(* CoDeSys 2.3.9.41 project: 25_06_aspiNEW.pro *)
(* Libraries: STANDARD.LIB 4.10.05 11:14:46, IECSFC.LIB 13.4.06 15:51:28, ANALYZATION.LIB 5.10.99 09:05:06 *)

(* PLC configuration (modules and I/O channels)
xDI_Start_F1 AT %IX0.0 [BitInput] Discrete input 1 {ChannellName = Enter name}
xDI_Stop_F1 AT %IX0.1 [BitInput] Discrete input 2 {ChannellName = Enter name}
xDI_Start_F2 AT %IX0.2 [BitInput] Discrete input 3 {ChannellName = Enter name}
xDI_Stop_F2 AT %IX0.3 [BitInput] Discrete input 4 {ChannellName = Enter name}
AT %IB1.0 [ByteInput] 8 discrete inputs {ChannellName = Enter name}
AT %IB1.1 [ByteInput] 8 discrete inputs {ChannellName = Enter name}
AT %IB1.2 [ByteInput] 8 discrete inputs {ChannellName = Enter name}
AT %IB1.3 [ByteInput] 8 discrete inputs {ChannellName = Enter name}
AT %QX2.0 [BitOutput] Fast discrete output 1 {ChannellName = Enter name}
AT %QX2.1 [BitOutput] Fast discrete output 2 {ChannellName = Enter name}
AT %QX2.2 [BitOutput] Fast discrete output 3 {ChannellName = Enter name}
xDO_Lamp_F1 AT %QX2.3 [BitOutput] Fast discrete output 4 {ChannellName = Enter name}
AT %QB3.0 [ByteOutput] 8 discrete outputs {ChannellName = Enter name}
AT %QB3.1 [ByteOutput] 8 discrete outputs {ChannellName = Enter name}
AT %QB3.2 [ByteOutput] 4 discrete outputs {ChannellName = Enter name}
Special input [ID103] node 4, in %IB4 out %QB4 {ChannellName = Special input}
  AT %IX4.0 [BitInput] Special input {ChannellName = Enter name}
Special output [ID104] node 5, in %IB5 out %QB5 {ChannellName = Special output}
  AT %QX5.0 [BitOutput] Special output {ChannellName = Enter name}
TCP [TCP_ID221] node 0, in %IB6.0.0 out %QB6.0.0 {ChannellName = TCP; RemotePort = 502; Visibility = No}
AT %QB6.1.0 [ByteOutput] {ChannellName = Enter name}
AT %QB6.2.0 [ByteOutput] {ChannellName = Enter name}
AT %QB6.3.0 [ByteOutput] {ChannellName = Enter name}
AT %QB6.4.0 [ByteOutput] {ChannellName = Enter name}
AT %QB6.5.0 [ByteOutput] {ChannellName = Enter name}
AT %QB6.6.0 [ByteOutput] {ChannellName = Enter name}
AT %QB6.7.0 [ByteOutput] {ChannellName = Enter name}
uiDelay_SCR_s AT %QW6.8.0 [WordOutput] {ChannellName = Enter name}
uiDelay_FAN_s AT %QW6.9.0 [WordOutput] {ChannellName = Enter name}
uiVib_Work_s AT %QW6.10.0 [WordOutput] {ChannellName = Enter name}
uiVib_Pause_min AT %QW6.11.0 [WordOutput] {ChannellName = Enter name}
uiHatch_Max_s AT %QW6.12.0 [WordOutput] {ChannellName = Enter name}
uiDrive_SpeedTimeout_s AT %QW6.13.0 [WordOutput] {ChannellName = Enter name}
uiFansRunning AT %QW6.14.0 [WordOutput] {ChannellName = Enter name}
uiModeDisplay AT %QW6.15.0 [WordOutput] {ChannellName = Enter name}
*)

(* Global variable list: GVL_AlarmIdx *)
VAR_GLOBAL CONSTANT
	ALM_EMERGENCY       : INT := 1;
	ALM_PRESSURE        : INT := 2;
	ALM_TF_DRIVE        : INT := 3;
	ALM_EXHAUST_DRIVE   : INT := 4;
	ALM_SCR_DRIVE       : INT := 5;
	ALM_SCR_IMPOSSIBLE  : INT := 7;
	ALM_F1_DRIVE        : INT := 10;
	ALM_F2_DRIVE        : INT := 11;
	ALM_F3_DRIVE        : INT := 12;
	ALM_F4_DRIVE        : INT := 13;
	ALM_F5_DRIVE        : INT := 14;
	ALM_VIB1            : INT := 20;
	ALM_VIB2            : INT := 21;
	ALM_HATCH 		: INT := 22;
	ALM_HATCH_TIMEOUT   : INT := 23;
END_VAR

(* Global variable list: GVL_App *)
VAR_GLOBAL
	(* === Исполнительные механизмы === *)
	TF		: ST_Motor;					(* Транспортный вентилятор *)
	Exhaust : ST_Motor;					(*Вытяжка*)
	SCR		: ST_Motor;					(* Шнек *)
	Fans	: ARRAY[1..5] OF ST_Fan;	(* Вентиляторы станков 1..5 *)
	Vib		: ST_Vibrator;				(* Пара вибраторов *)
	Hatch	: ST_Hatch;					(* Люк *)
	
	(* === Состояние системы === *)
	Alarms		: ST_Alarms;
	xModeManual	: BOOL;		(* Режим: FALSE = автомат, TRUE = ручной *)
	xAckAlarm	: BOOL;		(* Квитирование аварии (с панели) *)
	xMasterOK	: BOOL;		(* Магистраль готова (ТВ + шнек работают штатно) *)
END_VAR

(* Global variable list: GVL_HMI *)
VAR_GLOBAL RETAIN
	Settings : ST_Settings := (
		uiDelay_SCR_s          := 5,
		uiDelay_FAN_s          := 3,
		uiVib_Work_s           := 10,
		uiVib_Pause_min        := 30,
		uiHatch_Max_s          := 30,
		uiDrive_SpeedTimeout_s := 15	(* НОВОЕ *)
	);
END_VAR

(* Global variable list: GVL_Test *)
VAR_GLOBAL
	(* === Аварии === *)
	mb_Emergency      : BOOL;
	mb_Pressure       : BOOL;
	mb_TF_Alarm       : BOOL;
	mb_Exhaust_Alarm  : BOOL;
	mb_SCR_Alarm      : BOOL;
	mb_SCR_Impossible : BOOL;
	mb_Fan1_Alarm  : BOOL;
	mb_Fan2_Alarm  : BOOL;
	mb_Fan3_Alarm  : BOOL;
	mb_Fan4_Alarm  : BOOL;
	mb_Fan5_Alarm  : BOOL;
	mb_Vib1_Alarm  : BOOL;
	mb_Vib2_Alarm  : BOOL;
	mb_Hatch_Alarm   : BOOL;
	mb_Hatch_Timeout : BOOL;
END_VAR

(* Data type *)
TYPE E_DriveState :
(
	DRIVE_STOPPED  := 0,
	DRIVE_STARTING := 1,
	DRIVE_RUNNING  := 2,
	DRIVE_STOPPING := 3,
	DRIVE_FAULT    := 10
);
END_TYPE

(* Data type *)
TYPE E_HatchState :
(
	HATCH_UNKNOWN := 0,
	HATCH_CLOSED  := 1,
	HATCH_OPENING := 2,
	HATCH_OPEN    := 3,
	HATCH_CLOSING := 4,
	HATCH_FAULT   := 10
);
END_TYPE

(* Data type *)
TYPE E_VibState :
(
	VIB_IDLE	:= 0,	(* Выключено (xEnable=FALSE) *)
	VIB_PAUSE	:= 1,	(* Пауза между циклами *)
	VIB_WORK	:= 2	(* Фаза работы *)
);
END_TYPE

(* Data type *)
TYPE ST_Alarms :
STRUCT
	(* Критические *)
	xEmergencyStop  : BOOL;
	xPressure       : BOOL;
	xTF_Alarm       : BOOL;
	xExhaust_Alarm  : BOOL;
	xSCR_Alarm      : BOOL;
	xSCR_Impossible : BOOL;
	(* Предупреждения *)
	axFan_Alarm     : ARRAY[1..5] OF BOOL;
	xVib1_Alarm     : BOOL;
	xVib2_Alarm     : BOOL;
	xHatch_Alarm : BOOL;
	xHatch_Timeout  : BOOL;
	(* Обобщённые *)
	xAny      : BOOL;
	xCritical : BOOL;
	xWarning  : BOOL;
END_STRUCT
END_TYPE

(* Data type *)
TYPE ST_Fan :
STRUCT
    (* === Команды (вход в FB) === *)
 	xCmdStart    : BOOL;    (* Команда пуска (с кнопки или с панели) *)
	xCmdStop     : BOOL;    (* Команда стопа *)

	(* === Сигналы с поля (вход в FB) === *)
	xReady       : BOOL;    (* "Готов" от частотника (DI_readyF1) *)
	xAtSpeed  : BOOL;    (* "Авария" от частотника (DI_alarmF1) *)

	(* === Выход на ИМ === *)
	xRun         : BOOL;    (* Команда на пуск частотника (DO_F1) *)

	(* === Состояние (выход FB) === *)
	xEnabled     : BOOL;    (* Зафиксирован запрос на работу (был xFlag1) *)
	xFault       : BOOL;    (* Обобщённая неисправность (заменяет F1_OFF) *)
	eState       : E_DriveState;  (* Состояние машины: Stopped/Starting/Running/Fault *)

	(* === Статистика === *)
	udiStarts    : UDINT;   (* Счётчик пусков *)
	rHours       : REAL;    (* Моточасы *)
END_STRUCT
END_TYPE

(* Data type *)
TYPE ST_Hatch :
STRUCT
	(* === Команды === *)
	xCmdOpen      : BOOL;	(* Команда "Открыть" (удержание) *)
	xCmdClose     : BOOL;	(* Команда "Закрыть" (удержание) *)

	(* === Сигналы с поля === *)
	xLS_Open      : BOOL;	(* Концевик "Открыт" (DI33) *)
	xLS_Closed    : BOOL;	(* Концевик "Закрыт" (DI34) *)
	xAlarmHM      : BOOL;	(* Авария двигателя шибера (DI31) *)

	(* === Выходы на ИМ === *)
	xOpen         : BOOL;	(* DO "Открыть" (DO18) *)
	xClose        : BOOL;	(* DO "Закрыть" (DO19) *)

	(* === Состояние === *)
	eState        : E_HatchState;
	xFaultTimeout : BOOL;	(* Заклинило — таймаут *)
	xFault        : BOOL;	(* Обобщённая *)
END_STRUCT
END_TYPE

(* Data type *)
TYPE ST_Motor :
STRUCT
	(* === Команды (вход в FB) === *)
	xCmdRun		: BOOL;		(* Запрос на работу от секвенсора *)
	
	(* === Сигналы с поля === *)
	xReady		: BOOL;		(* "Готов" от частотника *)
	xAtSpeed	: BOOL;		(* "Авария" от частотника *)
	xRotation	: BOOL;		(* Импульсы датчика вращения (только для шнека) *)
	
	(* === Выход на ИМ === *)
	xRun		: BOOL;		(* Команда на пуск частотника *)
	
	(* === Состояние === *)
	xFault		: BOOL;		(* Обобщённая неисправность *)
	xNoRotation	: BOOL;		(* Авария "Не вращается" (только для шнека) *)
	eState		: E_DriveState;
END_STRUCT
END_TYPE

(* Data type *)
TYPE ST_Settings :
STRUCT
	(* === Тайминги секвенсора, секунды === *)
	uiDelay_SCR_s		: UINT;		(* Задержка пуска шнека после ТВ *)
	uiDelay_FAN_s		: UINT;		(* Задержка пуска вентилятора после шнека *)
	
	(* === Тайминги вибраторов === *)
	uiVib_Work_s		: UINT;		(* Длительность работы, секунды *)
	uiVib_Pause_min		: UINT;		(* Пауза между циклами, минуты *)
	
	(* === Тайминги люка === *)
	uiHatch_Max_s		: UINT;		(* Макс. время хода до концевика, секунды *)
	
	(* === Контроль шнека === *)
	uiScr_Window_s		: UINT;		(* Окно контроля вращения, секунды *)
	uiScr_PulseMin		: UINT;		(* Мин. импульсов за окно *)

	uiDrive_SpeedTimeout_s : UINT;
END_STRUCT
END_TYPE

(* Data type *)
TYPE ST_Vibrator :
STRUCT
	(* === Команды === *)
	xEnable		: BOOL;		(* Разрешение работы (от секвенсора: шнек работает) *)
	
	(* === Сигналы с поля === *)
	xAlarmV1	: BOOL;		(* Авария вибратора 1 *)
	xAlarmV2	: BOOL;		(* Авария вибратора 2 *)
	
	(* === Выходы на ИМ === *)
	xRunV1		: BOOL;
	xRunV2		: BOOL;
	
	(* === Состояние === *)
	xFault		: BOOL;
	xActive		: BOOL;		(* Сейчас идёт фаза работы (не паузы) *)
END_STRUCT
END_TYPE

(* POU PLC_PRG, ST *)
PROGRAM PLC_PRG
VAR
	(* === FB основных механизмов === *)
	FB_TF       : FB_Motor;
	FB_Exhaust  : FB_Motor;
	FB_SCR      : FB_Motor;
	FB_Fans     : ARRAY[1..5] OF FB_Fan;
	FB_Hatch    : FB_Hatch;
	FB_Vibrator : FB_Vibrator;
	FB_Alarms   : ARRAY[1..30] OF FB_Alarm;

	(* === Таймеры === *)
	TON_SCR_Delay : TON;
	TON_SCR_OffDelay : TON;	(* задержка выключения шнека *)
	TON_TF_OffDelay  : TON;	(* задержка выключения ТВ *)
	xAnyFanEnabled   : BOOL;	(* есть хоть один запрошенный вентилятор *)

	(* === Локальные массивы-агрегаторы команд === *)
	axCmdStart   : ARRAY[1..5] OF BOOL;
	axCmdStop    : ARRAY[1..5] OF BOOL;
	(*axAlarmDrive : ARRAY[1..5] OF BOOL;*)
	axAtSpeed :ARRAY[1..5] OF BOOL;
	axHMI_Man_Fan : ARRAY[1..5] OF BOOL;

	(* === Индекс цикла === *)
	i : INT;

	(* === Локальные копии TIME-настроек === *)
	tFanDelay  : TIME;
	tScrDelay  : TIME;
	tHatchMax  : TIME;
	tVibWork   : TIME;
	tVibPause  : TIME;
	tSpeedTimeout : TIME;

	(* === Флаги взаимной блокировки шибер <-> ИМ === *)
	xHatchClosed : BOOL;
	xAllStopped  : BOOL;

	xSettingsInit : BOOL;

	TON_Blink1 : TON;
	TON_Blink2 : TON;
	xBlink     : BOOL;
END_VAR
Inputs();
Diagnostics();
Sequence();
Outputs();
HMI();
ModbusMap();
END_PROGRAM
ACTION Diagnostics:
(* === КРИТИЧЕСКИЕ === *)
FB_Alarms[ALM_EMERGENCY](xCause := xDI_AlarmRelay, xAck := xAckAlarm);
Alarms.xEmergencyStop := FB_Alarms[ALM_EMERGENCY].xActive;

(* НЗ-контакт: норма = 24В (TRUE), авария/обрыв = нет 24В (FALSE) *)
FB_Alarms[ALM_PRESSURE](xCause := NOT xDI_Pressure, xAck := xAckAlarm);
Alarms.xPressure := FB_Alarms[ALM_PRESSURE].xActive;

(*FB_Alarms[ALM_TF_DRIVE](xCause := xDI_Alarm_TF, xAck := xAckAlarm);*)
FB_Alarms[ALM_TF_DRIVE](xCause := TF.xFault, xAck := xAckAlarm);
Alarms.xTF_Alarm := FB_Alarms[ALM_TF_DRIVE].xActive;

FB_Alarms[ALM_EXHAUST_DRIVE](xCause := xDI_Alarm_Exhaust, xAck := xAckAlarm);
Alarms.xExhaust_Alarm := FB_Alarms[ALM_EXHAUST_DRIVE].xActive;

(*FB_Alarms[ALM_SCR_DRIVE](xCause := xDI_Alarm_SCR, xAck := xAckAlarm);*)
FB_Alarms[ALM_SCR_DRIVE](xCause := SCR.xFault, xAck := xAckAlarm);
Alarms.xSCR_Alarm := FB_Alarms[ALM_SCR_DRIVE].xActive;

FB_Alarms[ALM_SCR_IMPOSSIBLE](xCause := NOT xDI_SCR_Impossible, xAck := xAckAlarm);
Alarms.xSCR_Impossible := FB_Alarms[ALM_SCR_IMPOSSIBLE].xActive;

(* === ВЕНТИЛЯТОРЫ 1..5 === *)
FB_Alarms[ALM_F1_DRIVE](xCause := Fans[1].xFault, xAck := xAckAlarm);
FB_Alarms[ALM_F2_DRIVE](xCause := Fans[2].xFault, xAck := xAckAlarm);
FB_Alarms[ALM_F3_DRIVE](xCause := Fans[3].xFault, xAck := xAckAlarm);
FB_Alarms[ALM_F4_DRIVE](xCause := Fans[4].xFault, xAck := xAckAlarm);
FB_Alarms[ALM_F5_DRIVE](xCause := Fans[5].xFault, xAck := xAckAlarm);

Alarms.axFan_Alarm[1] := FB_Alarms[ALM_F1_DRIVE].xActive;
Alarms.axFan_Alarm[2] := FB_Alarms[ALM_F2_DRIVE].xActive;
Alarms.axFan_Alarm[3] := FB_Alarms[ALM_F3_DRIVE].xActive;
Alarms.axFan_Alarm[4] := FB_Alarms[ALM_F4_DRIVE].xActive;
Alarms.axFan_Alarm[5] := FB_Alarms[ALM_F5_DRIVE].xActive;

(* === ВИБРАТОРЫ === *)
FB_Alarms[ALM_VIB1](xCause := xDI_Alarm_V1, xAck := xAckAlarm);
Alarms.xVib1_Alarm := FB_Alarms[ALM_VIB1].xActive;

FB_Alarms[ALM_VIB2](xCause := xDI_Alarm_V2, xAck := xAckAlarm);
Alarms.xVib2_Alarm := FB_Alarms[ALM_VIB2].xActive;

(* === ШИБЕР === *)
FB_Alarms[ALM_HATCH](xCause := xDI_Alarm_Hatch, xAck := xAckAlarm);
Alarms.xHatch_Alarm := FB_Alarms[ALM_HATCH].xActive;

FB_Alarms[ALM_HATCH_TIMEOUT](xCause := Hatch.xFaultTimeout, xAck := xAckAlarm);
Alarms.xHatch_Timeout := FB_Alarms[ALM_HATCH_TIMEOUT].xActive;

(* === КРИТИЧНЫЕ аварии: запрещают пуск всего, красный + зуммер === *)
Alarms.xCritical :=
	Alarms.xEmergencyStop                  (* аварийный стоп *)
	OR Alarms.xPressure                    (* нет разрежения *)
	OR Alarms.xSCR_Impossible              (* переполнение шнека *)
	OR FB_Alarms[ALM_TF_DRIVE].xActive     (* ТВ не набрал обороты — критично *)
	OR FB_Alarms[ALM_SCR_DRIVE].xActive;   (* шнек не набрал обороты — критично *)

(* === ПРЕДУПРЕЖДЕНИЯ: некритичные, жёлтый, система работает === *)
Alarms.xWarning :=
	FB_Alarms[ALM_F1_DRIVE].xActive
	OR FB_Alarms[ALM_F2_DRIVE].xActive
	OR FB_Alarms[ALM_F3_DRIVE].xActive
	OR FB_Alarms[ALM_F4_DRIVE].xActive
	OR FB_Alarms[ALM_F5_DRIVE].xActive
	OR FB_Alarms[ALM_VIB1].xActive
	OR FB_Alarms[ALM_VIB2].xActive
	OR FB_Alarms[ALM_HATCH].xActive;

Alarms.xAny := Alarms.xCritical OR Alarms.xWarning;

(* === СВЕТОФОР И ЗУММЕР === *)
IF Alarms.xCritical THEN
	xDO_Green  := FALSE;
	xDO_Yellow := FALSE;
	xDO_Red    := TRUE;
	xDO_Buzzer := TRUE;
ELSIF Alarms.xWarning OR NOT xDI_LS_Closed THEN
	xDO_Green  := FALSE;
	xDO_Yellow := TRUE;
	xDO_Red    := FALSE;
	xDO_Buzzer := FALSE;
ELSE
	xDO_Green  := TRUE;
	xDO_Yellow := FALSE;
	xDO_Red    := FALSE;
	xDO_Buzzer := FALSE;
END_IF
END_ACTION
ACTION HMI:
(* Сброс импульсных команд (кнопки вентиляторов) *)
xHMI_Start_F1 := FALSE;
xHMI_Start_F2 := FALSE;
xHMI_Start_F3 := FALSE;
xHMI_Start_F4 := FALSE;
xHMI_Start_F5 := FALSE;

xHMI_Stop_F1 := FALSE;
xHMI_Stop_F2 := FALSE;
xHMI_Stop_F3 := FALSE;
xHMI_Stop_F4 := FALSE;
xHMI_Stop_F5 := FALSE;

xHMI_AckAlarm := FALSE;
END_ACTION
ACTION Inputs:
(* Управление вентиляторами *)
axCmdStart[1] := xDI_Start_F1 OR xHMI_Start_F1;
axCmdStart[2] := xDI_Start_F2 OR xHMI_Start_F2;
axCmdStart[3] := xDI_Start_F3 OR xHMI_Start_F3;
axCmdStart[4] := xDI_Start_F4 OR xHMI_Start_F4;
axCmdStart[5] := xDI_Start_F5 OR xHMI_Start_F5;

axCmdStop[1] := xDI_Stop_F1 OR xHMI_Stop_F1;
axCmdStop[2] := xDI_Stop_F2 OR xHMI_Stop_F2;
axCmdStop[3] := xDI_Stop_F3 OR xHMI_Stop_F3;
axCmdStop[4] := xDI_Stop_F4 OR xHMI_Stop_F4;
axCmdStop[5] := xDI_Stop_F5 OR xHMI_Stop_F5;

(* Аварии частотников вентиляторов *)
(*
axAlarmDrive[1] := xDI_Alarm_F1;
axAlarmDrive[2] := xDI_Alarm_F2;
axAlarmDrive[3] := xDI_Alarm_F3;
axAlarmDrive[4] := xDI_Alarm_F4;
axAlarmDrive[5] := xDI_Alarm_F5;
*)

axAtSpeed[1] := xDI_AtSpeed_F1;
axAtSpeed[2] := xDI_AtSpeed_F2;
axAtSpeed[3] := xDI_AtSpeed_F3;
axAtSpeed[4] := xDI_AtSpeed_F4;
axAtSpeed[5] := xDI_AtSpeed_F5;

(* Команды на шибер *)
IF xModeManual THEN
	Hatch.xCmdOpen  := xHMI_Man_Open;
	Hatch.xCmdClose := xHMI_Man_Close;
ELSE
	Hatch.xCmdOpen  := xDI_Open  OR xHMI_Open;
	Hatch.xCmdClose := xDI_Close OR xHMI_Close;
END_IF

(* Сервисные сигналы *)
xAckAlarm   := xHMI_AckAlarm;
xModeManual := xHMI_ModeManual;

(* Ручные toggle вентиляторов -> в массив для цикла *)
axHMI_Man_Fan[1] := xHMI_Man_F1;
axHMI_Man_Fan[2] := xHMI_Man_F2;
axHMI_Man_Fan[3] := xHMI_Man_F3;
axHMI_Man_Fan[4] := xHMI_Man_F4;
axHMI_Man_Fan[5] := xHMI_Man_F5;
END_ACTION
ACTION ModbusMap:
(* ============================================================
   Action: ModbusMap — "промежуточные реле" для Modbus
   Копирование значений из структур в плоские переменные,
   т.к. конфигуратор ПЛК 2.3 не привязывает поля структур.
   Только ЧТЕНИЕ структур -> запись в mb_* (состояния на панель).
   ============================================================ *)

(* В начало ModbusMap *)
IF NOT xSettingsInit THEN
	IF uiDelay_SCR_s = 0 AND uiDelay_FAN_s = 0 THEN
		uiDelay_SCR_s   := 5;
		uiDelay_FAN_s   := 3;
		uiVib_Work_s    := 10;
		uiVib_Pause_min := 30;
		uiHatch_Max_s   := 30;
	END_IF
	xSettingsInit := TRUE;
END_IF

(* Работа механизмов *)
mb_Fan1_Run    := Fans[1].xRun;
mb_Fan2_Run    := Fans[2].xRun;
mb_Fan3_Run    := Fans[3].xRun;
mb_Fan4_Run    := Fans[4].xRun;
mb_Fan5_Run    := Fans[5].xRun;
mb_TF_Run      := TF.xRun;
mb_SCR_Run     := SCR.xRun;
mb_Exhaust_Run := Exhaust.xRun;

(* Вибраторы, магистраль, концевики *)
mb_Vib1_Run    := Vib.xRunV1;
mb_Vib2_Run    := Vib.xRunV2;
mb_Vib_Active  := Vib.xActive;
mb_MasterOK    := xMasterOK;
mb_LS_Open     := xDI_LS_Open;
mb_LS_Closed   := xDI_LS_Closed;
mb_Hatch_Open  := Hatch.xOpen;
mb_Hatch_Close := Hatch.xClose;

(* Аварии *)
mb_Emergency      := Alarms.xEmergencyStop;
mb_Pressure       := Alarms.xPressure;
mb_TF_Alarm       := Alarms.xTF_Alarm;
mb_Exhaust_Alarm  := Alarms.xExhaust_Alarm;
mb_SCR_Alarm      := Alarms.xSCR_Alarm;
mb_SCR_Impossible := Alarms.xSCR_Impossible;
mb_Fan1_Alarm  := Alarms.axFan_Alarm[1];
mb_Fan2_Alarm  := Alarms.axFan_Alarm[2];
mb_Fan3_Alarm  := Alarms.axFan_Alarm[3];
mb_Fan4_Alarm  := Alarms.axFan_Alarm[4];
mb_Fan5_Alarm  := Alarms.axFan_Alarm[5];
mb_Vib1_Alarm  := Alarms.xVib1_Alarm;
mb_Vib2_Alarm  := Alarms.xVib2_Alarm;
mb_Hatch_Alarm := Alarms.xHatch_Alarm;
mb_Hatch_Timeout := Alarms.xHatch_Timeout;
END_ACTION
ACTION Outputs:
(* ТВ, вытяжка и шнек *)
xDO_Run_TF      := TF.xRun;
xDO_Run_Exhaust := Exhaust.xRun;
xDO_Run_SCR     := SCR.xRun;

(* Вентиляторы 1..5 *)
xDO_Run_F1 := Fans[1].xRun;
xDO_Run_F2 := Fans[2].xRun;
xDO_Run_F3 := Fans[3].xRun;
xDO_Run_F4 := Fans[4].xRun;
xDO_Run_F5 := Fans[5].xRun;

(* Лампы у станков — по факту физической работы *)
xDO_Lamp_F1 := Fans[1].xRun;
xDO_Lamp_F2 := Fans[2].xRun;
xDO_Lamp_F3 := Fans[3].xRun;
xDO_Lamp_F4 := Fans[4].xRun;
xDO_Lamp_F5 := Fans[5].xRun;
(* Вибраторы *)
xDO_Run_V1 := Vib.xRunV1;
xDO_Run_V2 := Vib.xRunV2;

(* Шибер *)
xDO_HatchOpen  := Hatch.xOpen;
xDO_HatchClose := Hatch.xClose;

(* === Светосигнальная колонна === *)
(* Генератор мигания 1 Гц для зуммера *)
TON_Blink1(IN := NOT TON_Blink2.Q, PT := T#500MS);
TON_Blink2(IN := TON_Blink1.Q, PT := T#500MS);
xBlink := TON_Blink1.Q;

xDO_Red    := Alarms.xCritical;                              (* критично — красный *)
xDO_Yellow := Alarms.xWarning AND NOT Alarms.xCritical;      (* предупреждение — жёлтый *)
xDO_Green  := NOT Alarms.xCritical AND NOT Alarms.xWarning;  (* норма — зелёный *)

xDO_Buzzer := Alarms.xCritical AND xBlink;                   (* зуммер прерывисто при критичной *)
END_ACTION
ACTION Sequence:
(* 1. Конвертация настроек *)
tFanDelay  := DWORD_TO_TIME(UINT_TO_DWORD(uiDelay_FAN_s) * 1000);
tScrDelay  := DWORD_TO_TIME(UINT_TO_DWORD(uiDelay_SCR_s) * 1000);
tHatchMax  := DWORD_TO_TIME(UINT_TO_DWORD(uiHatch_Max_s) * 1000);
tVibWork   := DWORD_TO_TIME(UINT_TO_DWORD(uiVib_Work_s) * 1000);
tVibPause  := DWORD_TO_TIME(UINT_TO_DWORD(uiVib_Pause_min) * 60000);

(* === Таймаут набора оборотов ПЧ === *)
tSpeedTimeout := DWORD_TO_TIME(UINT_TO_DWORD(Settings.uiDrive_SpeedTimeout_s) * 1000);

(* === Clamp настроек (защита от битых значений) === *)
IF Settings.uiDelay_SCR_s < 1 THEN Settings.uiDelay_SCR_s := 1; END_IF
IF Settings.uiDelay_SCR_s > 30 THEN Settings.uiDelay_SCR_s := 30; END_IF
IF Settings.uiDelay_FAN_s < 1 THEN Settings.uiDelay_FAN_s := 1; END_IF
IF Settings.uiDelay_FAN_s > 30 THEN Settings.uiDelay_FAN_s := 30; END_IF
IF Settings.uiVib_Work_s < 5 THEN Settings.uiVib_Work_s := 5; END_IF
IF Settings.uiVib_Work_s > 120 THEN Settings.uiVib_Work_s := 120; END_IF
IF Settings.uiVib_Pause_min < 1 THEN Settings.uiVib_Pause_min := 1; END_IF
IF Settings.uiVib_Pause_min > 240 THEN Settings.uiVib_Pause_min := 240; END_IF
IF Settings.uiHatch_Max_s < 5 THEN Settings.uiHatch_Max_s := 5; END_IF
IF Settings.uiHatch_Max_s > 120 THEN Settings.uiHatch_Max_s := 120; END_IF
IF Settings.uiDrive_SpeedTimeout_s < 5 THEN Settings.uiDrive_SpeedTimeout_s := 5; END_IF
IF Settings.uiDrive_SpeedTimeout_s > 60 THEN Settings.uiDrive_SpeedTimeout_s := 60; END_IF

(* 2. Условия взаимной блокировки шибер <-> ИМ *)
(* ИМ разрешены только при полностью закрытом шибере *)
xHatchClosed := xDI_LS_Closed;

(* Шибер можно двигать только когда ВСЕ ИМ остановлены *)
xAllStopped :=
	NOT TF.xRun
	AND NOT SCR.xRun
	AND NOT Exhaust.xRun
	AND NOT Fans[1].xRun AND NOT Fans[2].xRun AND NOT Fans[3].xRun
	AND NOT Fans[4].xRun AND NOT Fans[5].xRun
	AND NOT Vib.xRunV1 AND NOT Vib.xRunV2;

(* 3. Магистраль готова? *)
xMasterOK := (TF.eState = DRIVE_RUNNING) AND (SCR.eState = DRIVE_RUNNING);

(* 4. Вентиляторы 1..5 *)
FOR i := 1 TO 5 DO
	FB_Fans[i](
		xCmdStart    := axCmdStart[i] AND NOT xModeManual,
		xCmdStop     := axCmdStop[i],
		(*xAlarmDrive  := Alarms.axFan_Alarm[i],*)
		xAtSpeed := axAtSpeed[i],
		xResetFault  := xAckAlarm,
		xMasterOK    := xMasterOK,
		xSystemFault := Alarms.xCritical OR NOT xHatchClosed,
		tStartDelay  := tFanDelay,
		tSpeedTimeout := tSpeedTimeout
	);

	IF xModeManual THEN
		(* Ручной режим: прямое управление toggle с защитами *)
		Fans[i].xRun :=
			axHMI_Man_Fan[i]
			AND NOT Alarms.axFan_Alarm[i]
			AND NOT Alarms.xEmergencyStop
			AND xHatchClosed;
		Fans[i].xEnabled := axHMI_Man_Fan[i];
		Fans[i].xFault   := FB_Fans[i].xFault;
		Fans[i].eState   := FB_Fans[i].eState;
	ELSE
		(* Автоматический режим: через FB_Fan *)
		Fans[i].xRun     := FB_Fans[i].xRun;
		Fans[i].xEnabled := FB_Fans[i].xEnabled;
		Fans[i].xFault   := FB_Fans[i].xFault;
		Fans[i].eState   := FB_Fans[i].eState;
	END_IF
END_FOR

(* ============================================================
   Управление ТВ и шнеком: пуск и обратный останов с паузами
   ============================================================ *)
IF xModeManual THEN
	(* Ручной режим — прямое управление с панели *)
	TF.xCmdRun  := xHMI_Man_TF  AND NOT Alarms.xTF_Alarm  AND NOT Alarms.xEmergencyStop AND xHatchClosed;
	SCR.xCmdRun := xHMI_Man_SCR AND NOT Alarms.xSCR_Alarm AND NOT Alarms.xEmergencyStop AND xHatchClosed;
	(* Сброс всех таймеров последовательности *)
	TON_SCR_Delay(IN := FALSE);
	TON_SCR_OffDelay(IN := FALSE);
	TON_TF_OffDelay(IN := FALSE);
ELSE
	(* === Автоматический режим === *)

	(* Есть ли хоть один запрошенный вентилятор *)
	xAnyFanEnabled :=
		Fans[1].xEnabled OR Fans[2].xEnabled OR Fans[3].xEnabled
		OR Fans[4].xEnabled OR Fans[5].xEnabled;

	(* --- ТРАНСПОРТНЫЙ ВЕНТИЛЯТОР --- *)
	(* Пуск: сразу как появился запрос вентилятора.
	   Останов: держим ещё, пока идёт цепочка останова (шнек + пауза TF). *)
	(* Таймер задержки ВЫКЛЮЧЕНИЯ ТВ: считает после выключения шнека *)
	TON_TF_OffDelay(IN := NOT SCR.xCmdRun AND NOT xAnyFanEnabled, PT := tScrDelay);

	TF.xCmdRun :=
		(xAnyFanEnabled OR SCR.xCmdRun OR NOT TON_TF_OffDelay.Q)
		AND NOT Alarms.xCritical
		AND xHatchClosed;

	(* --- ШНЕК --- *)
	(* Пуск: через паузу tScrDelay ПОСЛЕ выхода ТВ на режим.
	   Останов: через паузу tFanDelay ПОСЛЕ ухода последнего вентилятора. *)

	(* Таймер задержки ПУСКА шнека *)
	TON_SCR_Delay(
		IN := (TF.eState = DRIVE_RUNNING) AND xAnyFanEnabled AND NOT Alarms.xCritical,
		PT := tScrDelay
	);

	(* Таймер задержки ВЫКЛЮЧЕНИЯ шнека (после ухода последнего вентилятора) *)
	TON_SCR_OffDelay(IN := NOT xAnyFanEnabled, PT := tFanDelay);

	(* Команда шнеку:
	   - включается когда прошла пауза пуска (TON_SCR_Delay.Q)
	   - держится пока есть вентиляторы ИЛИ ещё идёт пауза останова (NOT TON_SCR_OffDelay.Q)
	   - гасится когда вентиляторов нет И прошла пауза останова *)
	IF NOT Alarms.xCritical AND (TF.eState = DRIVE_RUNNING) THEN
		IF xAnyFanEnabled THEN
			(* Фаза работы/пуска: включаем после паузы пуска *)
			IF TON_SCR_Delay.Q THEN
				SCR.xCmdRun := TRUE;
			END_IF
		ELSE
			(* Фаза останова: держим пока не прошла пауза выключения *)
			IF TON_SCR_OffDelay.Q THEN
				SCR.xCmdRun := FALSE;
			END_IF
		END_IF
	ELSE
		SCR.xCmdRun := FALSE;
	END_IF
END_IF

(* 6. FB_Motor для ТВ *)
FB_TF(
	xCmdRun     := TF.xCmdRun,
	(*xAlarmDrive := xDI_Alarm_TF,*)
	xAtSpeed      := xDI_AtSpeed_TF,
	xResetFault := xAckAlarm,
	tSpeedTimeout := tSpeedTimeout
);
TF.xRun   := FB_TF.xRun;
TF.xFault := FB_TF.xFault;
TF.eState := FB_TF.eState;

(* 7. FB_Motor для шнека *)
FB_SCR(
	xCmdRun     := SCR.xCmdRun,
	(*xAlarmDrive := xDI_Alarm_SCR,*)
	xAtSpeed      := xDI_AtSpeed_SCR,
	xResetFault := xAckAlarm,
	tSpeedTimeout := tSpeedTimeout
);
SCR.xRun   := FB_SCR.xRun;
SCR.xFault := FB_SCR.xFault;
SCR.eState := FB_SCR.eState;

(* 8. Вытяжка *)
FB_Exhaust(
	xCmdRun     := xHMI_Exhaust AND NOT Alarms.xEmergencyStop AND xHatchClosed,
	xAtSpeed := xDI_Alarm_Exhaust,
	xResetFault := xAckAlarm,
);
Exhaust.xRun   := FB_Exhaust.xRun;
Exhaust.xFault := FB_Exhaust.xFault;
Exhaust.eState := FB_Exhaust.eState;

(* 9. Вибраторы *)
FB_Vibrator(
	xEnable  := (SCR.eState = DRIVE_RUNNING) AND NOT xModeManual AND NOT Alarms.xCritical,
	xAlarmV1 := xDI_Alarm_V1,
	xAlarmV2 := xDI_Alarm_V2,
	tWork    := tVibWork,
	tPause   := tVibPause
);
IF xModeManual THEN
	Vib.xRunV1 := xHMI_Man_V1 AND NOT Alarms.xVib1_Alarm AND NOT Alarms.xEmergencyStop AND xHatchClosed;
	Vib.xRunV2 := xHMI_Man_V2 AND NOT Alarms.xVib2_Alarm AND NOT Alarms.xEmergencyStop AND xHatchClosed;
ELSE
	Vib.xRunV1 := FB_Vibrator.xRunV1;
	Vib.xRunV2 := FB_Vibrator.xRunV2;
END_IF
Vib.xFault  := FB_Vibrator.xFault;
Vib.xActive := FB_Vibrator.xActive;

(* 10. Шибер — движение только когда всё остановлено *)
FB_Hatch(
	xCmdOpen    := Hatch.xCmdOpen  AND xAllStopped,
	xCmdClose   := Hatch.xCmdClose AND xAllStopped,
	xLS_Open    := xDI_LS_Open,
	xLS_Closed  := xDI_LS_Closed,
	xAlarmHatch := xDI_Alarm_Hatch,
	xResetFault := xAckAlarm,
	tMaxTravel  := tHatchMax
);
Hatch.xOpen         := FB_Hatch.xOpen;
Hatch.xClose        := FB_Hatch.xClose;
Hatch.eState        := FB_Hatch.eState;
Hatch.xFault        := FB_Hatch.xFault;
Hatch.xFaultTimeout := FB_Hatch.xFaultTimeout;

(* === Критичная авария: стоп всей магистрали === *)
IF Alarms.xCritical THEN
	TF.xCmdRun  := FALSE;
	SCR.xCmdRun := FALSE;
	FOR i := 1 TO 5 DO
		axCmdStart[i] := FALSE;	(* снять запросы пуска вентиляторов *)
	END_FOR
END_IF
END_ACTION

(* POU FB_Motor, ST *)
FUNCTION_BLOCK FB_Motor
VAR_INPUT
	xCmdRun     : BOOL;
	xAtSpeed : BOOL;
	xResetFault : BOOL;
	tSpeedTimeout : TIME;
END_VAR
VAR_OUTPUT
	xRun   : BOOL;
	xFault : BOOL;
	eState : E_DriveState;
END_VAR
VAR
	TON_Speed : TON;
END_VAR
(* Авария привода (ПЧ или защита контактора) -> FAULT *)
IF xAtSpeed THEN
	IF eState = DRIVE_FAULT THEN
		eState := DRIVE_STOPPED;
	END_IF
END_IF

(* Сброс аварии по квитированию, если причина устранена *)
(*IF xResetFault AND NOT xAlarmDrive THEN
	IF eState = DRIVE_FAULT THEN
		eState := DRIVE_STOPPED;
	END_IF
END_IF
*)

(* Машина состояний *)
CASE eState OF
	DRIVE_STOPPED:
		xRun := FALSE;
		TON_Speed(IN := FALSE);

		(*IF xCmdRun AND NOT xAlarmDrive THEN
			eState := DRIVE_RUNNING;
		END_IF *)

		IF xCmdRun THEN
			eState := DRIVE_RUNNING;
		END_IF
	DRIVE_RUNNING :
		xRun := TRUE;
		TON_Speed(IN := NOT xAtSpeed, PT := tSpeedTimeout);
		IF NOT xCmdRun THEN
			eState := DRIVE_STOPPED;
		ELSIF TON_Speed.Q THEN
			eState := DRIVE_FAULT;
		END_IF
	DRIVE_FAULT:
		xRun := FALSE;
		TON_Speed(IN := FALSE);
END_CASE

xFault := (eState = DRIVE_FAULT);
END_FUNCTION_BLOCK

(* POU FB_Fan, ST *)
FUNCTION_BLOCK FB_Fan
VAR_INPUT
	xCmdStart    : BOOL;
	xCmdStop     : BOOL;
	xAtSpeed       : BOOL;
	xResetFault  : BOOL;
	xMasterOK    : BOOL;
	xSystemFault : BOOL;
	tStartDelay  : TIME;
	tSpeedTimeout : TIME;
END_VAR
VAR_OUTPUT
	xRun     : BOOL;
	xEnabled : BOOL;
	xFault   : BOOL;
	eState   : E_DriveState;
END_VAR
VAR
	RS_Cmd         : RS;
	TON_StartDelay : TON;
	TON_Speed      : TON;
	(* xMasterWasReady : BOOL;	 магистраль была готова уже при запросе *)
END_VAR
(* 1. Фиксация команды пуска.
   Команда сбрасывается при Stop, аварии привода или системной аварии *)
RS_Cmd(
	SET := xCmdStart,
	RESET1 := xCmdStop OR xSystemFault
);
xEnabled := RS_Cmd.Q1;

(* 2. Авария привода -> переход в FAULT *)
(*IF xAlarmDrive THEN
	eState := DRIVE_FAULT;
END_IF *)

(* Сброс аварии по квитированию, если причина устранена *)
IF xResetFault AND NOT xAtSpeed THEN
	IF eState = DRIVE_FAULT THEN
		eState := DRIVE_STOPPED;
	END_IF
END_IF

(* 3. Машина состояний *)
CASE eState OF
	DRIVE_STOPPED:
		xRun := FALSE;
		TON_StartDelay(IN := FALSE);
		IF xEnabled AND NOT xSystemFault THEN
			(* Запоминаем: магистраль уже работает? *)
			(*xMasterWasReady := xMasterOK;*)
			eState := DRIVE_STARTING;
		END_IF

	DRIVE_STARTING:
		xRun := FALSE;
		(*IF NOT xEnabled OR xSystemFault THEN
			eState := DRIVE_STOPPED;
		ELSIF xMasterWasReady THEN
			(* Магистраль уже работала на момент запроса — пуск без задержки *)
			eState := DRIVE_RUNNING;
		ELSE
			(* Магистраль раскручивается — ждём готовности + выдержку *)
			TON_StartDelay(IN := xMasterOK, PT := tStartDelay);
			IF TON_StartDelay.Q THEN
				eState := DRIVE_RUNNING;
			END_IF *)
		TON_StartDelay(IN := xMasterOK, PT := tStartDelay);
		TON_Speed(IN := FALSE);
		IF NOT xEnabled OR xSystemFault THEN
			eState := DRIVE_STOPPED;
		ELSIF TON_StartDelay.Q THEN
			eState := DRIVE_RUNNING;
		END_IF

	DRIVE_RUNNING:
		xRun := TRUE;
		TON_Speed(IN := NOT xAtSpeed, PT := tSpeedTimeout);
		IF NOT xEnabled OR xSystemFault OR NOT xMasterOK THEN
			eState := DRIVE_STOPPED;
		ELSIF TON_Speed.Q THEN
			eState := DRIVE_FAULT;	(* за 15с не набрал обороты *)
		END_IF

	DRIVE_FAULT:
		xRun := FALSE;
		TON_Speed(IN := FALSE);
END_CASE

(* 4. Обобщённая неисправность *)
xFault := (eState = DRIVE_FAULT);
END_FUNCTION_BLOCK

(* POU FB_Hatch, ST *)
FUNCTION_BLOCK FB_Hatch
VAR_INPUT
	xCmdOpen    : BOOL;
	xCmdClose   : BOOL;
	xLS_Open    : BOOL;
	xLS_Closed  : BOOL;
	xAlarmHatch    : BOOL;
	xResetFault : BOOL;
	tMaxTravel  : TIME;
END_VAR
VAR_OUTPUT
	xOpen         : BOOL;
	xClose        : BOOL;
	eState        : E_HatchState;
	xFaultTimeout : BOOL;
	xFault        : BOOL;
END_VAR
VAR
	TON_Travel : TON;
END_VAR
(* Авария двигателя шибера -> FAULT *)
IF xAlarmHatch THEN
	eState := HATCH_FAULT;
END_IF

(* Сброс аварии по квитированию *)
IF xResetFault AND NOT xAlarmHatch THEN
	IF eState = HATCH_FAULT THEN
		eState := HATCH_UNKNOWN;
		xFaultTimeout := FALSE;
	END_IF
END_IF

(* Движение по удержанию кнопки. Приоритет "Закрыть" *)
IF eState = HATCH_FAULT THEN
	xOpen  := FALSE;
	xClose := FALSE;
	TON_Travel(IN := FALSE);

ELSIF xCmdClose THEN
	(* Закрытие: едем пока кнопка удержана И не сработал концевик "закрыт" *)
	xOpen  := FALSE;
	xClose := NOT xLS_Closed;
	eState := HATCH_CLOSING;
	TON_Travel(IN := xClose, PT := tMaxTravel);
	IF TON_Travel.Q THEN
		xFaultTimeout := TRUE;
		eState := HATCH_FAULT;
	END_IF

ELSIF xCmdOpen THEN
	(* Открытие: едем пока кнопка удержана И не сработал концевик "открыт" *)
	xClose := FALSE;
	xOpen  := NOT xLS_Open;
	eState := HATCH_OPENING;
	TON_Travel(IN := xOpen, PT := tMaxTravel);
	IF TON_Travel.Q THEN
		xFaultTimeout := TRUE;
		eState := HATCH_FAULT;
	END_IF

ELSE
	(* Кнопки отпущены — стоп, фиксируем положение по концевикам *)
	xOpen  := FALSE;
	xClose := FALSE;
	TON_Travel(IN := FALSE);
	IF xLS_Open THEN
		eState := HATCH_OPEN;
	ELSIF xLS_Closed THEN
		eState := HATCH_CLOSED;
	ELSE
		eState := HATCH_UNKNOWN;
	END_IF
END_IF

xFault := (eState = HATCH_FAULT);
END_FUNCTION_BLOCK

(* POU FB_Vibrator, ST *)
(* ============================================================
   FB_Vibrator — управление парой вибраторов фильтра
   
   Циклограмма (пока xEnable = TRUE):
   - При пуске: пауза tPause -> работа tWork -> пауза -> работа -> ...
   - Оба вибратора V1 и V2 включаются одновременно
   - Авария одного вибратора: не включаем его, второй работает
     (если у него нет аварии). Циклограмма не нарушается.
   - xEnable = FALSE -> немедленно стоп, сброс цикла
   ============================================================ *)
FUNCTION_BLOCK FB_Vibrator
VAR_INPUT
	xEnable		: BOOL;		(* Разрешение работы (шнек крутится) *)
	xAlarmV1	: BOOL;		(* Авария вибратора 1 *)
	xAlarmV2	: BOOL;		(* Авария вибратора 2 *)
	tWork		: TIME;		(* Длительность фазы работы *)
	tPause		: TIME;		(* Длительность паузы *)
END_VAR
VAR_OUTPUT
	xRunV1	: BOOL;			(* На физический выход V1 *)
	xRunV2	: BOOL;			(* На физический выход V2 *)
	xFault	: BOOL;			(* Есть авария хоть одного вибратора *)
	xActive	: BOOL;			(* Сейчас фаза работы (для индикации) *)
END_VAR
VAR
	eState		: E_VibState;
	TON_Pause	: TON;
	TON_Work	: TON;
END_VAR
(* ====================================================================
   Машина состояний циклограммы
   ==================================================================== *)
CASE eState OF
	
	VIB_IDLE:
		xRunV1	:= FALSE;
		xRunV2	:= FALSE;
		xActive	:= FALSE;
		TON_Pause(IN := FALSE);
		TON_Work(IN := FALSE);
		(* Запуск цикла — начинаем с паузы, чтобы вибраторы 
		   не включались сразу при пуске шнека *)
		IF xEnable THEN
			eState := VIB_PAUSE;
		END_IF
	
	VIB_PAUSE:
		xRunV1	:= FALSE;
		xRunV2	:= FALSE;
		xActive	:= FALSE;
		TON_Pause(IN := TRUE, PT := tPause);
		TON_Work(IN := FALSE);
		
		IF NOT xEnable THEN
			eState := VIB_IDLE;
		ELSIF TON_Pause.Q THEN
			TON_Pause(IN := FALSE);
			eState := VIB_WORK;
		END_IF
	
	VIB_WORK:
		(* Включаем только исправные вибраторы *)
		xRunV1	:= NOT xAlarmV1;
		xRunV2	:= NOT xAlarmV2;
		xActive	:= TRUE;
		TON_Pause(IN := FALSE);
		TON_Work(IN := TRUE, PT := tWork);
		
		IF NOT xEnable THEN
			eState := VIB_IDLE;
		ELSIF TON_Work.Q THEN
			TON_Work(IN := FALSE);
			eState := VIB_PAUSE;
		END_IF

END_CASE


(* ====================================================================
   Обобщённая авария (для жёлтой лампы)
   ==================================================================== *)
xFault := xAlarmV1 OR xAlarmV2;
END_FUNCTION_BLOCK

(* POU FB_Alarm, ST *)
(* ============================================================
   FB_Alarm — обработчик одной аварии с фиксацией и квитированием
   
   Поведение:
   - При появлении xCause -> xActive = TRUE (зафиксирована)
   - xActive остаётся TRUE, даже если xCause пропала
   - Сброс только при: xAck (квитирование) И xCause = FALSE
   - Это защищает от автоматического "самосброса" аварии
   ============================================================ *)
FUNCTION_BLOCK FB_Alarm
VAR_INPUT
	xCause	: BOOL;		(* Причина аварии (например, xDI_Alarm_TF) *)
	xAck	: BOOL;		(* Квитирование от оператора *)
END_VAR
VAR_OUTPUT
	xActive	: BOOL;		(* Авария активна (для индикации и блокировок) *)
END_VAR
VAR
	R_TRIG_Ack	: R_TRIG;	(* Фронт квитирования *)
END_VAR
(* Фронт квитирования — реагируем только на момент нажатия *)
R_TRIG_Ack(CLK := xAck);

(* Установка: причина появилась — авария зафиксирована *)
IF xCause THEN
	xActive := TRUE;
END_IF

(* Сброс: квитирование по фронту И причина устранена *)
IF R_TRIG_Ack.Q AND NOT xCause THEN
	xActive := FALSE;
END_IF
END_FUNCTION_BLOCK
